// TIA Portal V17 export
// export: Created 2023-06-23T18:33:38.9275153Z, ExportSetting WithDefaults, DisplayName Totally Integrated Automation Portal, DisplayVersion V17, DisplayName TIA Portal Openness, DisplayVersion V17, DisplayName TIA Portal Version Control Interface, DisplayVersion V17, DisplayName STEP 7 Professional, DisplayVersion V17, DisplayName STEP 7 Safety, DisplayVersion V17, DisplayName WinCC Advanced / Unified PC, DisplayVersion V17
VAR_GLOBAL   // PLC tag table "13_SC1-EXA"
   "iSC1-EXAp" AT %I8.5 : Bool;
   "iSC1-EXA" AT %I8.6 : Bool;
   "oSC1-EXAp" AT %Q8.0 : Bool;
   "oSC1-EXA" AT %Q8.1 : Bool;
END_VAR
